{attribute 'GeneratedUsingTerminal: EL1502-0000-0018'}
{attribute addProperty BoxType "EL1502-0000-0018"}
{attribute addProperty Id "StatusAT %I*Status_26C2D68E8Counter_valueAT %I*UDINT4"}
{attribute addProperty CRC "3066269297"}
{attribute addProperty Size "12"}
TYPE CNT_Inputs_B6C38E71 :
STRUCT
	{attribute addProperty Name "Status"}
	Status AT %I* : Status_26C2D68E;
	{attribute addProperty Name "Counter_value"}
	Counter_value AT %I* : UDINT;
END_STRUCT
END_TYPE

(* stored: Version 1.2.0.0, ProductVersion 3.1.4024.9
   DUT CNT_Inputs_B6C38E71: Id {2b3c4a56-ab1d-48dd-a1e6-8d4fd879a9b0} *)
